FUNCTION FC_HeaderCounters : UDINT
VAR_INPUT
    In: STRING(50);
	FindLeft : BOOL;
END_VAR
VAR
	tempString	: T_MaxString;
	Pos : INT;
END_VAR

Pos := FIND(In, '/');
IF FindLeft THEN
	tempString := LEFT(In, LEN(In)-Pos);
ELSE
	tempString := RIGHT(In, LEN(In)-Pos);
END_IF

FC_HeaderCounters := STRING_TO_UDINT(tempString);

END_FUNCTION

(* stored: Version 1.1.0.1, ProductVersion 3.1.4024.15
   POU FC_HeaderCounters: Id {ad4e63d2-4c92-42fa-989d-94dfcbd48fdc}, SpecialFunc None *)
